TYPE ST_3D_Values :
STRUCT
	X :REAL;
	Y :REAL;
	Z :REAL;
END_STRUCT
END_TYPE

(* stored: Version 1.1.0.1, ProductVersion 3.1.4024.13
   DUT ST_3D_Values: Id {5bb496d1-5e69-4190-a436-474b883bd44a} *)
